PROGRAM PRG_PLAS_17_MovePacksToOCVCtrl
VAR
	tonEnableCameraSystem					: TON;
	bEnableStackTriggeringAfterDelay			: BOOL;
	bEnableStackAggregationCameraSystem	: BOOL;

	tofStackConfirmationCameraOFFDelay 		: TOF;

	fbMoveOuterStatusArray					: FB_PACK_MoveOuterStatusArray;
	fbAddNewOCVTriggerID					: FB_PLAS_AddNewTriggerID;

	rtrigNewArrived						: R_TRIG;
	bNewCodeIsProccesing				: BOOL;

	fbCodeDiag					: FB_SCANNER_DiagnosticLog;

	tonValidationTimout					: TON;
	bValidationTimeout					: BOOL;
	bValidationTimeoutReset				: BOOL;

	fbStackConfirmationCamera			: FB_SCANNER_CameraSelect;
	fbStackAggregationEvaluation			: FB_SCANNER_Evaluation;

	rtStackConfirmationCameraDone		:  R_TRIG;
	bStackConfirmationCameraDone		:  BOOL;

	fbMoveDataToOCVStatus				: FB_T04_MoveDataToOCVStatus;
	sMoveDataLog							: STRING;

	ctuConsecutiveNoConfirmation		: CTU;
	nDaignosticConfirmationCount		: INT;

	fbDebugCNT				: FB_DEBUG_CounterArray;
	aCNTDebug				: ARRAY [1..10] OF UDINT;
	bResetCNT					: BOOL;

END_VAR
VAR // added by the converter: edge detectors and wires of the graphical bodies
    _w1 : BOOL;
END_VAR

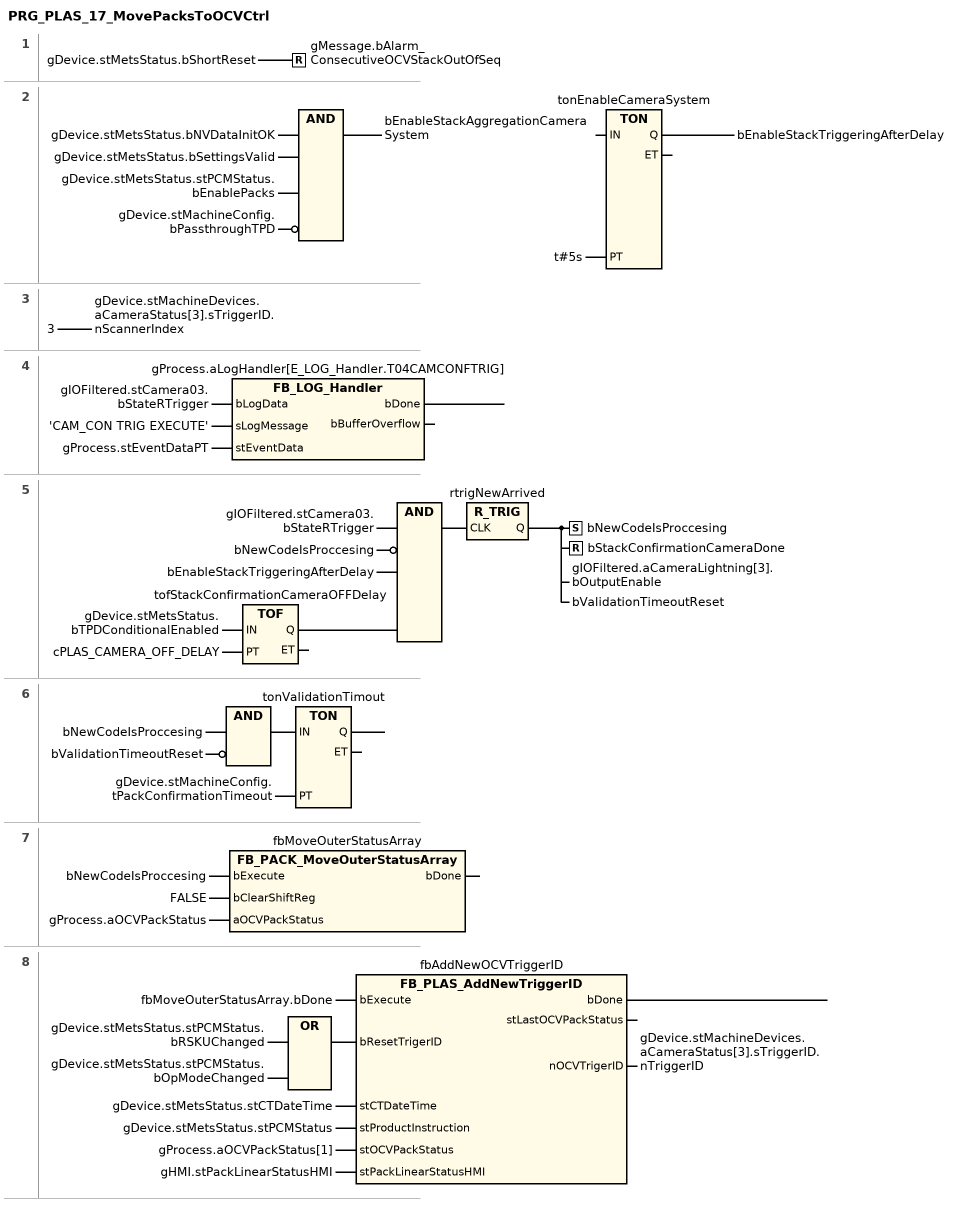
// NETWORK 1
gMessage.bAlarm_ConsecutiveOCVStackOutOfSeq R= gDevice.stMetsStatus.bShortReset;

// NETWORK 2
_w1 := gDevice.stMetsStatus.bNVDataInitOK AND gDevice.stMetsStatus.bSettingsValid AND gDevice.stMetsStatus.stPCMStatus.bEnablePacks AND NOT gDevice.stMachineConfig.bPassthroughTPD;
bEnableStackAggregationCameraSystem := _w1;
tonEnableCameraSystem(IN := _w1, PT := t#5s); // TON
bEnableStackTriggeringAfterDelay := tonEnableCameraSystem.Q;

// NETWORK 3
gDevice.stMachineDevices.aCameraStatus[3].sTriggerID.nScannerIndex := 3;

// NETWORK 4
gProcess.aLogHandler[E_LOG_Handler.T04CAMCONFTRIG](
    bLogData := gIOFiltered.stCamera03.bStateRTrigger,
    sLogMessage := 'CAM_CON TRIG EXECUTE',
    stEventData := gProcess.stEventDataPT); // FB_LOG_Handler

// NETWORK 5
tofStackConfirmationCameraOFFDelay(IN := gDevice.stMetsStatus.bTPDConditionalEnabled, PT := cPLAS_CAMERA_OFF_DELAY); // TOF
rtrigNewArrived(CLK := gIOFiltered.stCamera03.bStateRTrigger AND NOT bNewCodeIsProccesing AND bEnableStackTriggeringAfterDelay AND tofStackConfirmationCameraOFFDelay.Q); // R_TRIG
bNewCodeIsProccesing S= rtrigNewArrived.Q;
bStackConfirmationCameraDone R= rtrigNewArrived.Q;
gIOFiltered.aCameraLightning[3].bOutputEnable := rtrigNewArrived.Q;
bValidationTimeoutReset := rtrigNewArrived.Q;

// NETWORK 6
tonValidationTimout(IN := bNewCodeIsProccesing AND NOT bValidationTimeoutReset, PT := gDevice.stMachineConfig.tPackConfirmationTimeout); // TON

// NETWORK 7
fbMoveOuterStatusArray(
    bExecute := bNewCodeIsProccesing,
    bClearShiftReg := FALSE,
    aOCVPackStatus := gProcess.aOCVPackStatus); // FB_PACK_MoveOuterStatusArray

// NETWORK 8
fbAddNewOCVTriggerID(
    bExecute := fbMoveOuterStatusArray.bDone,
    bResetTrigerID := gDevice.stMetsStatus.stPCMStatus.bRSKUChanged OR gDevice.stMetsStatus.stPCMStatus.bOpModeChanged,
    stCTDateTime := gDevice.stMetsStatus.stCTDateTime,
    stProductInstruction := gDevice.stMetsStatus.stPCMStatus,
    stOCVPackStatus := gProcess.aOCVPackStatus[1],
    stPackLinearStatusHMI := gHMI.stPackLinearStatusHMI,
    nOCVTrigerID => gDevice.stMachineDevices.aCameraStatus[3].sTriggerID.nTriggerID); // FB_PLAS_AddNewTriggerID

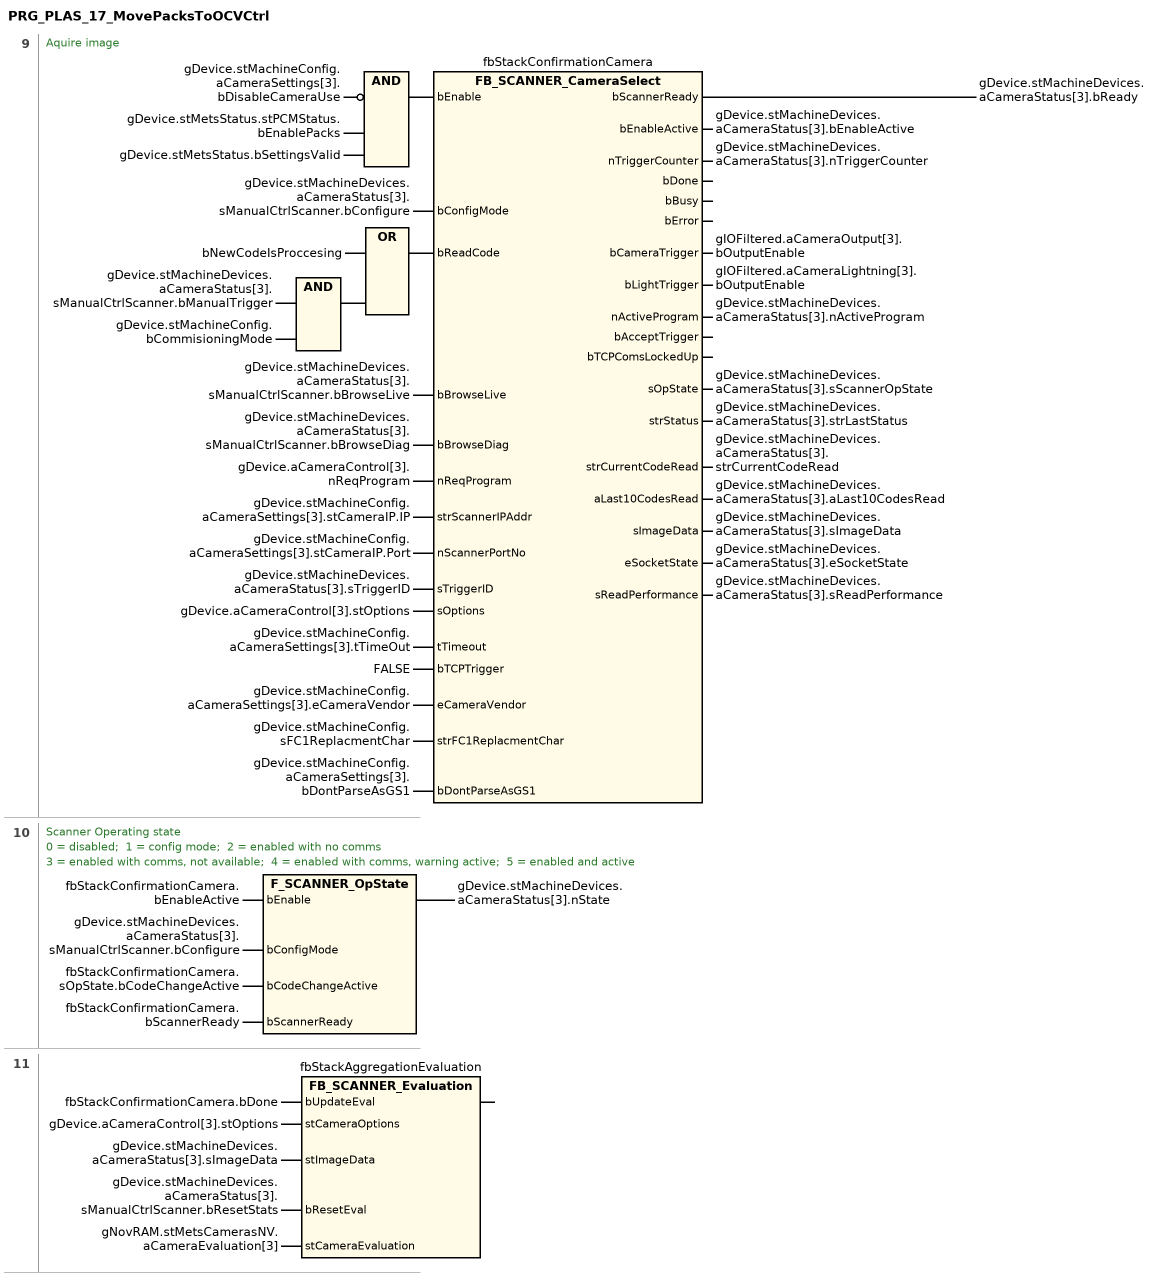
// NETWORK 9
// Aquire image
fbStackConfirmationCamera(
    bEnable := NOT gDevice.stMachineConfig.aCameraSettings[3].bDisableCameraUse AND gDevice.stMetsStatus.stPCMStatus.bEnablePacks AND gDevice.stMetsStatus.bSettingsValid,
    bConfigMode := gDevice.stMachineDevices.aCameraStatus[3].sManualCtrlScanner.bConfigure,
    bReadCode := bNewCodeIsProccesing OR gDevice.stMachineDevices.aCameraStatus[3].sManualCtrlScanner.bManualTrigger AND gDevice.stMachineConfig.bCommisioningMode,
    bBrowseLive := gDevice.stMachineDevices.aCameraStatus[3].sManualCtrlScanner.bBrowseLive,
    bBrowseDiag := gDevice.stMachineDevices.aCameraStatus[3].sManualCtrlScanner.bBrowseDiag,
    nReqProgram := gDevice.aCameraControl[3].nReqProgram,
    strScannerIPAddr := gDevice.stMachineConfig.aCameraSettings[3].stCameraIP.IP,
    nScannerPortNo := gDevice.stMachineConfig.aCameraSettings[3].stCameraIP.Port,
    sTriggerID := gDevice.stMachineDevices.aCameraStatus[3].sTriggerID,
    sOptions := gDevice.aCameraControl[3].stOptions,
    tTimeout := gDevice.stMachineConfig.aCameraSettings[3].tTimeOut,
    bTCPTrigger := FALSE,
    eCameraVendor := gDevice.stMachineConfig.aCameraSettings[3].eCameraVendor,
    strFC1ReplacmentChar := gDevice.stMachineConfig.sFC1ReplacmentChar,
    bDontParseAsGS1 := gDevice.stMachineConfig.aCameraSettings[3].bDontParseAsGS1,
    bEnableActive => gDevice.stMachineDevices.aCameraStatus[3].bEnableActive,
    nTriggerCounter => gDevice.stMachineDevices.aCameraStatus[3].nTriggerCounter,
    bCameraTrigger => gIOFiltered.aCameraOutput[3].bOutputEnable,
    bLightTrigger => gIOFiltered.aCameraLightning[3].bOutputEnable,
    nActiveProgram => gDevice.stMachineDevices.aCameraStatus[3].nActiveProgram,
    sOpState => gDevice.stMachineDevices.aCameraStatus[3].sScannerOpState,
    strStatus => gDevice.stMachineDevices.aCameraStatus[3].strLastStatus,
    strCurrentCodeRead => gDevice.stMachineDevices.aCameraStatus[3].strCurrentCodeRead,
    aLast10CodesRead => gDevice.stMachineDevices.aCameraStatus[3].aLast10CodesRead,
    sImageData => gDevice.stMachineDevices.aCameraStatus[3].sImageData,
    eSocketState => gDevice.stMachineDevices.aCameraStatus[3].eSocketState,
    sReadPerformance => gDevice.stMachineDevices.aCameraStatus[3].sReadPerformance); // FB_SCANNER_CameraSelect
gDevice.stMachineDevices.aCameraStatus[3].bReady := fbStackConfirmationCamera.bScannerReady;

// NETWORK 10
// 					Scanner Operating state
// 0 = disabled;  1 = config mode;  2 = enabled with no comms
// 3 = enabled with comms, not available;  4 = enabled with comms, warning active;  5 = enabled and active
//
gDevice.stMachineDevices.aCameraStatus[3].nState := F_SCANNER_OpState(bEnable := fbStackConfirmationCamera.bEnableActive, bConfigMode := gDevice.stMachineDevices.aCameraStatus[3].sManualCtrlScanner.bConfigure, bCodeChangeActive := fbStackConfirmationCamera.sOpState.bCodeChangeActive, bScannerReady := fbStackConfirmationCamera.bScannerReady);

// NETWORK 11
fbStackAggregationEvaluation(
    bUpdateEval := fbStackConfirmationCamera.bDone,
    stCameraOptions := gDevice.aCameraControl[3].stOptions,
    stImageData := gDevice.stMachineDevices.aCameraStatus[3].sImageData,
    bResetEval := gDevice.stMachineDevices.aCameraStatus[3].sManualCtrlScanner.bResetStats,
    stCameraEvaluation := gNovRAM.stMetsCamerasNV.aCameraEvaluation[3]); // FB_SCANNER_Evaluation

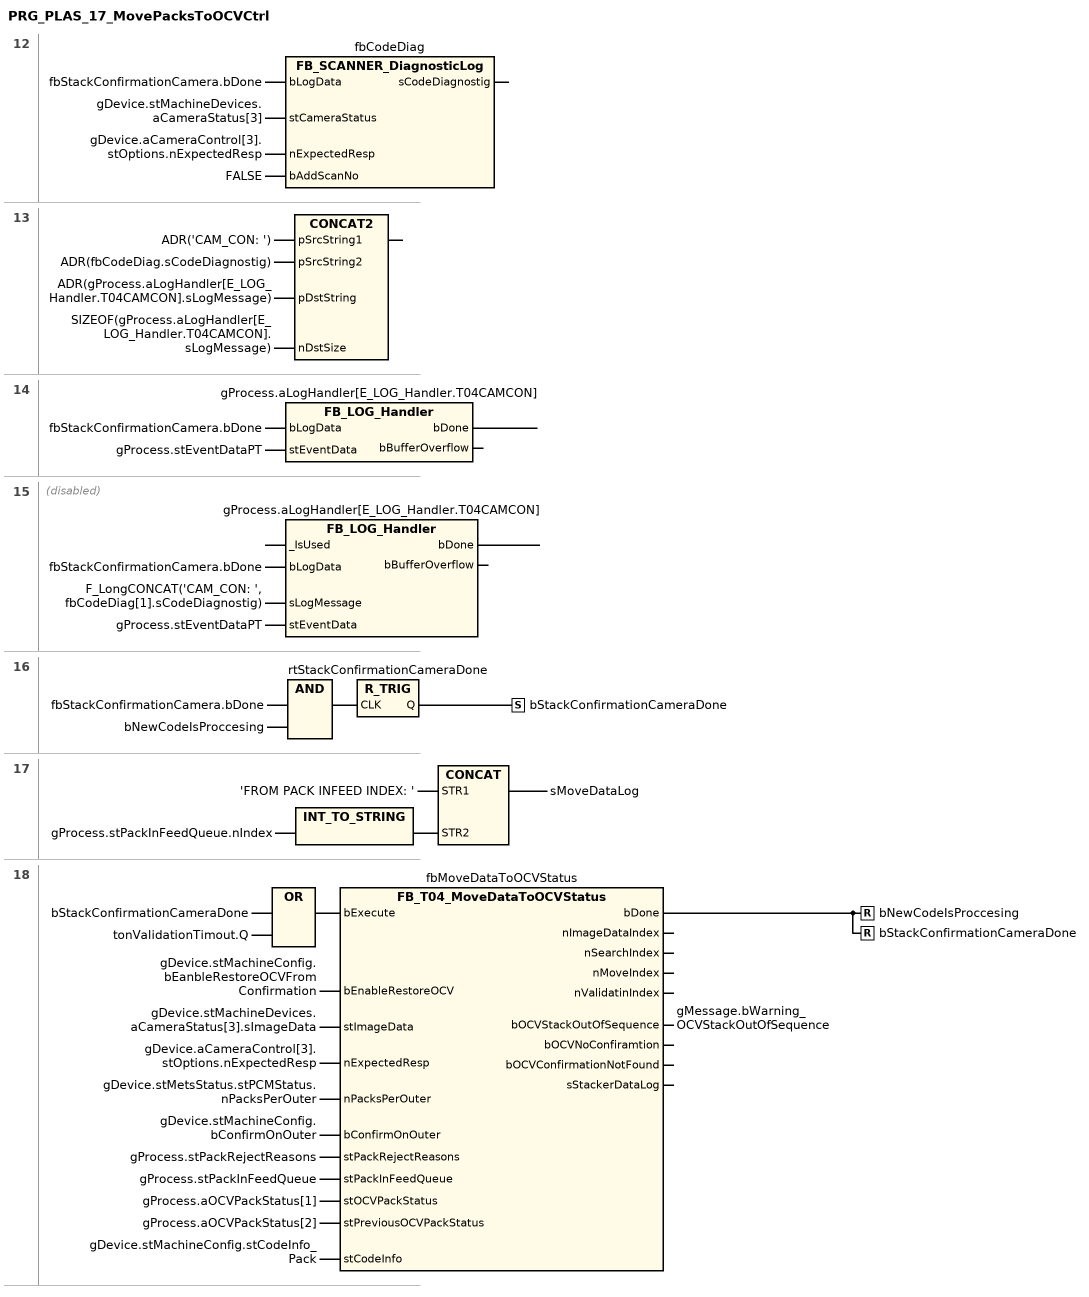
// NETWORK 12
fbCodeDiag(
    bLogData := fbStackConfirmationCamera.bDone,
    stCameraStatus := gDevice.stMachineDevices.aCameraStatus[3],
    nExpectedResp := gDevice.aCameraControl[3].stOptions.nExpectedResp,
    bAddScanNo := FALSE); // FB_SCANNER_DiagnosticLog

// NETWORK 13
CONCAT2(pSrcString1 := ADR('CAM_CON: '), pSrcString2 := ADR(fbCodeDiag.sCodeDiagnostig), pDstString := ADR(gProcess.aLogHandler[E_LOG_Handler.T04CAMCON].sLogMessage), nDstSize := SIZEOF(gProcess.aLogHandler[E_LOG_Handler.T04CAMCON].sLogMessage));

// NETWORK 14
gProcess.aLogHandler[E_LOG_Handler.T04CAMCON](bLogData := fbStackConfirmationCamera.bDone, stEventData := gProcess.stEventDataPT); // FB_LOG_Handler

// NETWORK 15 (disabled)
// gProcess.aLogHandler[E_LOG_Handler.T04CAMCON](
//     bLogData := fbStackConfirmationCamera.bDone,
//     sLogMessage := F_LongCONCAT('CAM_CON: ', fbCodeDiag[1].sCodeDiagnostig),
//     stEventData := gProcess.stEventDataPT); // FB_LOG_Handler

// NETWORK 16
rtStackConfirmationCameraDone(CLK := fbStackConfirmationCamera.bDone AND bNewCodeIsProccesing); // R_TRIG
bStackConfirmationCameraDone S= rtStackConfirmationCameraDone.Q;

// NETWORK 17
sMoveDataLog := CONCAT(STR1 := 'FROM PACK INFEED INDEX: ', STR2 := INT_TO_STRING(gProcess.stPackInFeedQueue.nIndex));

// NETWORK 18
fbMoveDataToOCVStatus(
    bExecute := bStackConfirmationCameraDone OR tonValidationTimout.Q,
    bEnableRestoreOCV := gDevice.stMachineConfig.bEanbleRestoreOCVFromConfirmation,
    stImageData := gDevice.stMachineDevices.aCameraStatus[3].sImageData,
    nExpectedResp := gDevice.aCameraControl[3].stOptions.nExpectedResp,
    nPacksPerOuter := gDevice.stMetsStatus.stPCMStatus.nPacksPerOuter,
    bConfirmOnOuter := gDevice.stMachineConfig.bConfirmOnOuter,
    stPackRejectReasons := gProcess.stPackRejectReasons,
    stPackInFeedQueue := gProcess.stPackInFeedQueue,
    stOCVPackStatus := gProcess.aOCVPackStatus[1],
    stPreviousOCVPackStatus := gProcess.aOCVPackStatus[2],
    stCodeInfo := gDevice.stMachineConfig.stCodeInfo_Pack,
    bOCVStackOutOfSequence => gMessage.bWarning_OCVStackOutOfSequence); // FB_T04_MoveDataToOCVStatus
bNewCodeIsProccesing R= fbMoveDataToOCVStatus.bDone;
bStackConfirmationCameraDone R= fbMoveDataToOCVStatus.bDone;

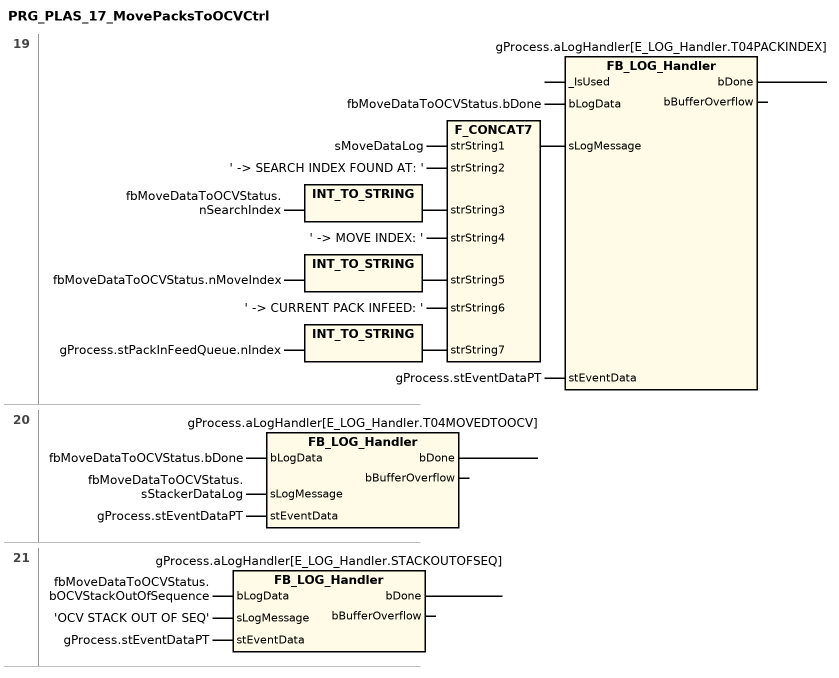
// NETWORK 19
gProcess.aLogHandler[E_LOG_Handler.T04PACKINDEX](
    bLogData := fbMoveDataToOCVStatus.bDone,
    sLogMessage := F_CONCAT7(strString1 := sMoveDataLog, strString2 := ' -> SEARCH INDEX FOUND AT: ', strString3 := INT_TO_STRING(fbMoveDataToOCVStatus.nSearchIndex), strString4 := ' -> MOVE INDEX: ', strString5 := INT_TO_STRING(fbMoveDataToOCVStatus.nMoveIndex), strString6 := ' -> CURRENT PACK INFEED: ', strString7 := INT_TO_STRING(gProcess.stPackInFeedQueue.nIndex)),
    stEventData := gProcess.stEventDataPT); // FB_LOG_Handler

// NETWORK 20
gProcess.aLogHandler[E_LOG_Handler.T04MOVEDTOOCV](
    bLogData := fbMoveDataToOCVStatus.bDone,
    sLogMessage := fbMoveDataToOCVStatus.sStackerDataLog,
    stEventData := gProcess.stEventDataPT); // FB_LOG_Handler

// NETWORK 21
gProcess.aLogHandler[E_LOG_Handler.STACKOUTOFSEQ](
    bLogData := fbMoveDataToOCVStatus.bOCVStackOutOfSequence,
    sLogMessage := 'OCV STACK OUT OF SEQ',
    stEventData := gProcess.stEventDataPT); // FB_LOG_Handler

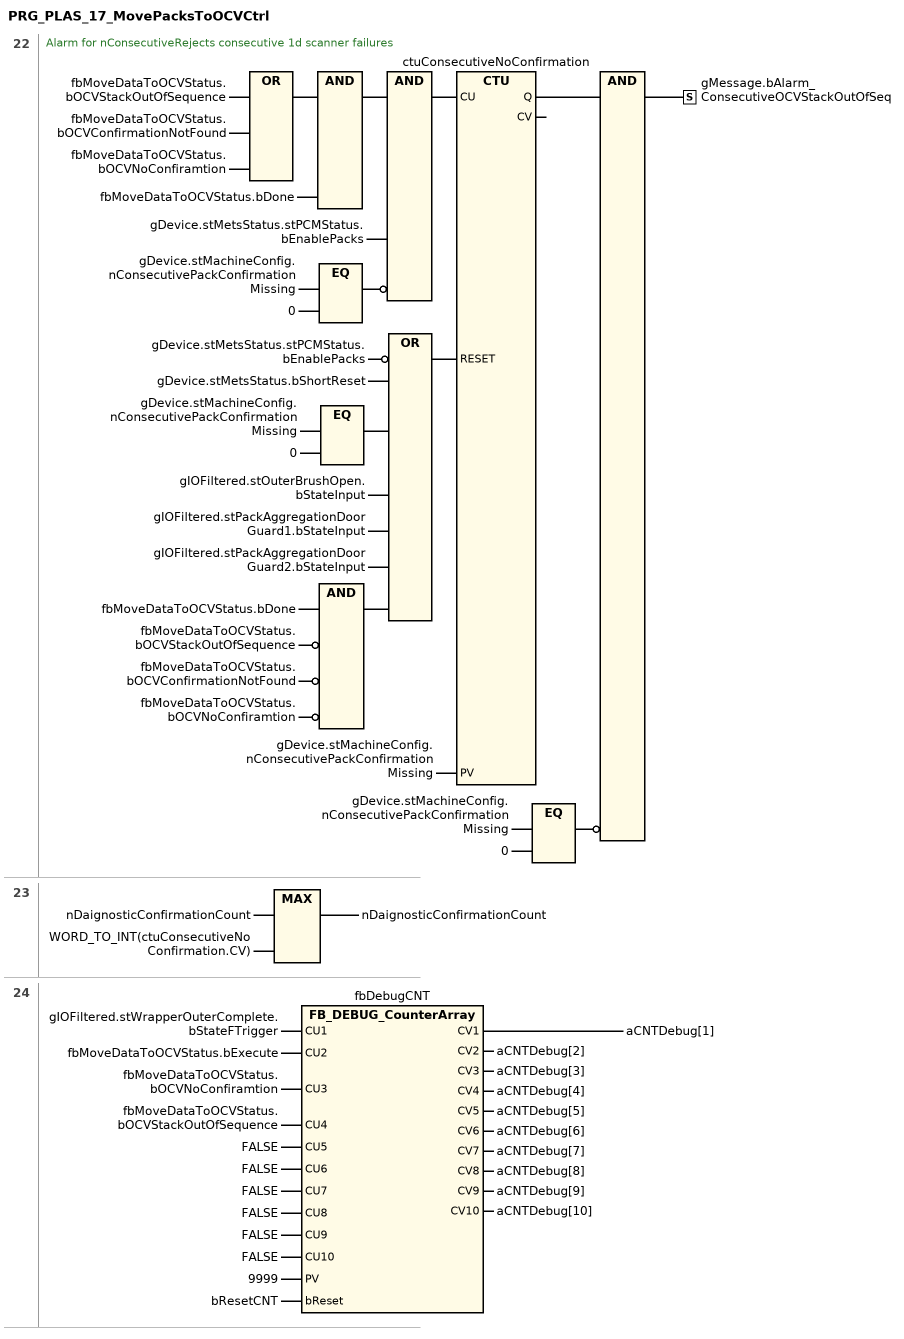
// NETWORK 22
// Alarm for nConsecutiveRejects consecutive 1d scanner failures
ctuConsecutiveNoConfirmation(
    CU := ((fbMoveDataToOCVStatus.bOCVStackOutOfSequence OR fbMoveDataToOCVStatus.bOCVConfirmationNotFound OR fbMoveDataToOCVStatus.bOCVNoConfiramtion) AND fbMoveDataToOCVStatus.bDone) AND gDevice.stMetsStatus.stPCMStatus.bEnablePacks AND NOT (gDevice.stMachineConfig.nConsecutivePackConfirmationMissing = 0),
    RESET := NOT gDevice.stMetsStatus.stPCMStatus.bEnablePacks OR gDevice.stMetsStatus.bShortReset OR gDevice.stMachineConfig.nConsecutivePackConfirmationMissing = 0 OR gIOFiltered.stOuterBrushOpen.bStateInput OR gIOFiltered.stPackAggregationDoorGuard1.bStateInput OR gIOFiltered.stPackAggregationDoorGuard2.bStateInput OR fbMoveDataToOCVStatus.bDone AND NOT fbMoveDataToOCVStatus.bOCVStackOutOfSequence AND NOT fbMoveDataToOCVStatus.bOCVConfirmationNotFound AND NOT fbMoveDataToOCVStatus.bOCVNoConfiramtion,
    PV := gDevice.stMachineConfig.nConsecutivePackConfirmationMissing); // CTU
gMessage.bAlarm_ConsecutiveOCVStackOutOfSeq S= ctuConsecutiveNoConfirmation.Q AND NOT (gDevice.stMachineConfig.nConsecutivePackConfirmationMissing = 0);

// NETWORK 23
nDaignosticConfirmationCount := MAX(nDaignosticConfirmationCount, WORD_TO_INT(ctuConsecutiveNoConfirmation.CV));

// NETWORK 24
fbDebugCNT(
    CU1 := gIOFiltered.stWrapperOuterComplete.bStateFTrigger,
    CU2 := fbMoveDataToOCVStatus.bExecute,
    CU3 := fbMoveDataToOCVStatus.bOCVNoConfiramtion,
    CU4 := fbMoveDataToOCVStatus.bOCVStackOutOfSequence,
    CU5 := FALSE,
    CU6 := FALSE,
    CU7 := FALSE,
    CU8 := FALSE,
    CU9 := FALSE,
    CU10 := FALSE,
    PV := 9999,
    bReset := bResetCNT,
    CV2 => aCNTDebug[2],
    CV3 => aCNTDebug[3],
    CV4 => aCNTDebug[4],
    CV5 => aCNTDebug[5],
    CV6 => aCNTDebug[6],
    CV7 => aCNTDebug[7],
    CV8 => aCNTDebug[8],
    CV9 => aCNTDebug[9],
    CV10 => aCNTDebug[10]); // FB_DEBUG_CounterArray
aCNTDebug[1] := fbDebugCNT.CV1;

END_PROGRAM

(* stored: Version 1.1.0.1
   POU PRG_PLAS_17_MovePacksToOCVCtrl: Id {c95455f8-1867-4a7f-9ad5-19236646ad48}, SpecialFunc None *)
